{attribute 'qualified_only'}
{attribute 'strict'}
TYPE eTypeOfTixon :
(
	TixonStep := 0,
	TixonVibro:=1,
	TixonPickStep:=2,
	TixonPickVibro:=3,
	TixonPickVibroBasic:=4
);
END_TYPE

(* stored: Version 1.1.0.1, ProductVersion 3.1.4024.12
   DUT eTypeOfTixon: Id {e72684ba-faa0-0269-3bf4-3a138c1c69a0} *)
